(* CoDeSys 2.3 export: PROC_ERR_STATUS.EXP *)

(* POU 60_Error handling/Process Errors/proc_Err_Status, ST *)
PROGRAM proc_Err_Status
VAR
	ProcessErr1_fb		: handleError;


END_VAR
;
END_PROGRAM
